Omron CX-Programmer project NewProject (CX-Programmer 9.75)

# PLC NewPLC1: CP1H XA

## Global symbols (name address type ; comment)
2.00 BOOL  ; Stop
1.00 BOOL  ; Start
100.00 BOOL  ; K1
101.00 BOOL  ; Y1
0.03 BOOL  ; CNT1
200.00 BOOL  ; K2
300.00 BOOL  ; C3
C0001 BOOL  ; C1
C0003 BOOL  ; CNT1
T0001 BOOL  ; T1
T0002 BOOL  ; T2

## Program NewProgram1 (cyclic task 0)
Local symbols
K1 BOOL
Start BOOL
Start1 BOOL

### Section Section1

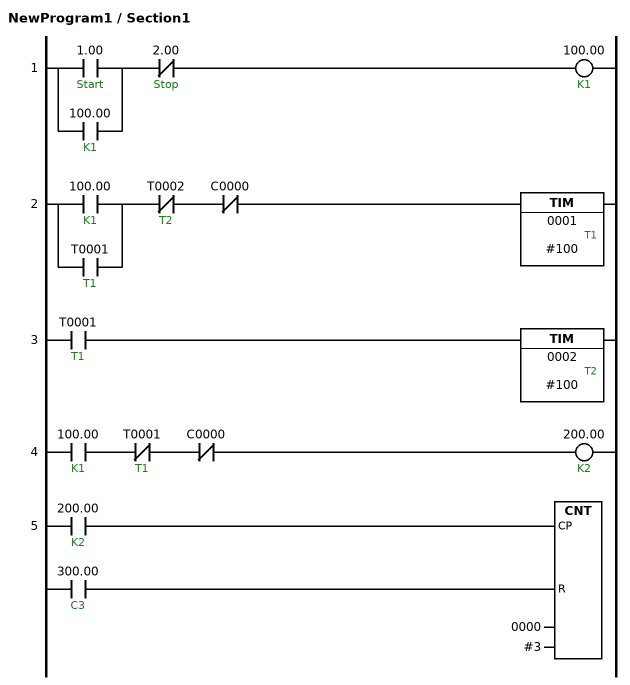
; rung 1
LD 1.00  ; Start
OR 100.00  ; K1
ANDNOT 2.00  ; Stop
OUT 100.00  ; K1
; rung 2
LD 100.00  ; K1
OR T0001  ; T1
ANDNOT T0002  ; T2
ANDNOT C0000
TIM 0001 #100  ; T1
; rung 3
LD T0001  ; T1
TIM 0002 #100  ; T2
; rung 4
LD 100.00  ; K1
ANDNOT T0001  ; T1
ANDNOT C0000
OUT 200.00  ; K2
; rung 5
LD 200.00  ; K2
LD 300.00  ; C3
CNT 0000 #3

### Section END
; rung 0
END(001)